(* CODESYS project collision_1.xml

Project tree, tasks and I/O mapping:
  function collision_1 [ST]
*)

// collision_1
FUNCTION collision_1 : BOOL
VAR_INPUT
END_VAR
VAR
END_VAR

IF collision_1 THEN
	collision_1	:=		FALSE;
END_IF

END_FUNCTION
